FUNCTION_BLOCK FB_PLCTPL_BASE
VAR_INPUT
	{attribute 'OPC.UA.DA':='0'}
	in_sName:				STRING	:= 'Shutter';	// Instance name

	{attribute 'OPC.UA.DA':='0'}
	in_bActiveLowClosed:	BOOL 	:= FALSE;		// If TRUE, the CLOSED signal is Active Low, default FALSE
	{attribute 'OPC.UA.DA':='0'}
	in_bActiveLowFault:		BOOL 	:= FALSE;		// If TRUE, the FAULT signal is Active Low, default FALSE
	{attribute 'OPC.UA.DA':='0'}
	in_bActiveLowOpen:		BOOL 	:= FALSE;		// If TRUE, the OPEN signal is Active Low, default FALSE
	{attribute 'OPC.UA.DA':='0'}
	in_bActiveLowSwitch:	BOOL 	:= FALSE;		// If TRUE, the SWITCH signal is Active Low, default FALSE

	{attribute 'OPC.UA.DA':='0'}
	in_bIgnoreClosed:		BOOL 	:= FALSE;		// If TRUE, the CLOSED signal is Ignored, default FALSE
	{attribute 'OPC.UA.DA':='0'}
	in_bIgnoreFault:		BOOL 	:= FALSE;		// If TRUE, the FAULT signal is Ignored, default FALSE
	{attribute 'OPC.UA.DA':='0'}
	in_bIgnoreOpen:			BOOL 	:= FALSE;		// If TRUE, the OPEN signal is Ignored, default FALSE

	
	{attribute 'OPC.UA.DA':='0'}
	in_bInitialState:		BOOL 	:= FALSE;		// Default shutter position is FALSE/CLOSED
	{attribute 'OPC.UA.DA':='0'}
	in_nTimeout:     		UDINT 	:= 3000;		// Timeout for OPEN/CLOSE transitions [msec], default 3000 ms

	{attribute 'OPC.UA.DA':='0'}
	in_bLogExtTime:			BOOL 	:= FALSE;		// If TRUE, use external time in event logs. Default FALSE.
	{attribute 'OPC.UA.DA':='0'}
	in_bLog:				BOOL 	:= TRUE;		// If TRUE, log events. Default TRUE.
END_VAR
VAR_OUTPUT
END_VAR
VAR RETAIN
END_VAR
VAR
	{attribute 'OPC.UA.DA' := '1'}
	cfg:		T_PLCTPL_CFG;	
	{attribute 'OPC.UA.DA' := '1'}
	ctrl:		T_PLCTPL_CTRL;	
	{attribute 'OPC.UA.DA' := '1'}
	{attribute 'OPC.UA.DA.Access' := '1'}
	info:		T_PLCTPL_INFO;	(* ReadOnly *)
	{attribute 'OPC.UA.DA' := '1'}
	{attribute 'OPC.UA.DA.Access' := '1'}
	stat:		T_PLCTPL_STAT;	(* ReadOnly *)

	{attribute 'OPC.UA.DA' := '0'}
	nEvent:		      	DINT := E_PLCTPL_EVENT.NONE;
	{attribute 'OPC.UA.DA' := '0'}
	nInternalEvent:		DINT := E_PLCTPL_EVENT.NONE;
	
	// Operational Events
	{attribute 'OPC.UA.DA' := '0'}
	fbEventStart:	FB_TcMessage;
	{attribute 'OPC.UA.DA' := '0'}
	fbEventEnd:		FB_TcMessage;
	{attribute 'OPC.UA.DA' := '0'}
	fbEventError:	FB_TcMessage;
	{attribute 'OPC.UA.DA' := '0'}
	fbEventDebug:	FB_TcMessage;
	{attribute 'OPC.UA.DA' := '0'}
	fbEventGeneral:	FB_TcMessage;
	
	(***** Physical signals - to be mapped!!! *****)

	(* Outputs *)

	(* Inputs *)
	
	// Flag if the device is ready to receive commands.
	// It takes a couple of cycles for the system to read inputs after reboot.
	{attribute 'OPC.UA.DA' := '0'}
	bDeviceReady:	BOOL 	:= FALSE;

END_VAR

// On first cycle configure from input params and internally execute M_UserConfigure()
IF NOT bDeviceReady THEN
	// Set device Configuration
	M_Configure();
	RETURN;
END_IF

// Increment counter.
// This will be seen as 'alive' flag.
stat.nCycleCounter	:= stat.nCycleCounter + 1;


(* === Check for commands and internal events to be processed === *)
CheckForEvents();

(* === Process events according to the State Machine === *)
ProcessEvents();

METHOD ActionCloseExecute
VAR_INPUT
END_VAR
END_METHOD

METHOD ActionDisableExecute
VAR_INPUT
END_VAR
END_METHOD

METHOD ActionEnableComplete
VAR_INPUT
END_VAR
END_METHOD

METHOD ActionEnableExecute
VAR_INPUT
END_VAR
END_METHOD

METHOD ActionErrExecute
VAR_INPUT
	nEventId:			DINT;
END_VAR
END_METHOD

METHOD ActionInitAbort
VAR_INPUT
END_VAR
END_METHOD

METHOD ActionInitComplete
VAR_INPUT
END_VAR
END_METHOD

METHOD ActionInitExecute
VAR_INPUT
END_VAR
END_METHOD

METHOD ActionInitReject
VAR_INPUT
END_VAR
END_METHOD

METHOD ActionOpenExecute
VAR_INPUT
END_VAR
END_METHOD

METHOD ActionResetExecute
VAR_INPUT
END_VAR
END_METHOD

METHOD ActionStopExecute
VAR_INPUT
END_VAR
END_METHOD

METHOD ActionUnexpExecute
VAR_INPUT
	nEventId:			DINT;
END_VAR
END_METHOD

METHOD ActivityClosing
VAR_INPUT
END_VAR
END_METHOD

METHOD ActivityDisabling
VAR_INPUT
END_VAR
END_METHOD

METHOD ActivityInitializing
VAR_INPUT
END_VAR
END_METHOD

METHOD ActivityOpening
VAR_INPUT
END_VAR
END_METHOD

METHOD CheckForEvents
VAR_INPUT
END_VAR
END_METHOD

METHOD M_Configure : BOOL
VAR_INPUT
END_VAR
VAR
     fbGetCurTaskIdx:	GETCURTASKINDEX;
END_VAR
// If device is ready, there is nothing to configure.
IF bDeviceReady THEN
	RETURN;
END_IF

// If first cycle, copy configuration AND RETURN in order for the system to read all inputs before doing any work
IF stat.nCycleCounter = 0 THEN
	cfg.sName				:= in_sName;			// Instance name
	cfg.bActiveLowClosed	:= in_bActiveLowClosed;	// If TRUE, the CLOSED signal is Active Low, default FALSE
	cfg.bActiveLowFault		:= in_bActiveLowFault;	// If TRUE, the FAULT signal is Active Low, default FALSE
	cfg.bActiveLowOpen		:= in_bActiveLowOpen;	// If TRUE, the OPEN signal is Active Low, default FALSE
	cfg.bActiveLowSwitch	:= in_bActiveLowSwitch;	// If TRUE, the SWITCH signal is Active Low, default FALSE

	cfg.bIgnoreClosed		:= in_bIgnoreClosed;	// If TRUE, the CLOSED signal is Ignored, default FALSE
	cfg.bIgnoreFault		:= in_bIgnoreFault;		// If TRUE, the FAULT signal is Ignored, default FALSE
	cfg.bIgnoreOpen			:= in_bIgnoreOpen;		// If TRUE, the OPEN signal is Ignored, default FALSE

	cfg.bInitialState		:= in_bInitialState;	// Default shutter position is FALSE/CLOSED
	cfg.nTimeout			:= in_nTimeout;			// Timeout for OPEN/CLOSE transitions [msec], default 3000 ms

	cfg.bLogExtTime			:= in_bLogExtTime;		// If TRUE, use external time in event logs
	cfg.bLog				:= in_bLog;				// If TRUE, use external time in event logs
	
	// Get the version number 
	stat.sLibVersion	:= Global_Version.stLibVersion_ESO_LDC_PLC_Template_Library.sVersion;

 	// Get cycle time in microsec.
	// CycleTime in _TaskInfo is given in 100 ns. 1 us = 1000 ns
	fbGetCurTaskIdx();
	stat.nCycleTime	:=  (TwinCAT_SystemInfoVarList._TaskInfo[fbGetCurTaskIdx.index].CycleTime)/10;
	
	// Increment counter.
	stat.nCycleCounter	:= stat.nCycleCounter + 1;
	RETURN;
ELSIF (stat.nCycleCounter * stat.nCycleTime) < 5000000 THEN
	// EtherCAT is normally ready after 3.5 sec.
	// We give it 5 sec to consider it to be ready.
	// Increment counter.
	stat.nCycleCounter	:= stat.nCycleCounter + 1;
	RETURN;
END_IF

// The system shoud be ready, i.e. coupler state is 8.

// Create Event instances
fbEventStart.CreateEx	(TC_EVENTS.plctplOpsEventClass.ActionStart,0);
fbEventEnd.CreateEx		(TC_EVENTS.plctplOpsEventClass.ActionEnd,0);
fbEventError.CreateEx	(TC_EVENTS.plctplOpsEventClass.Error,0);
fbEventDebug.CreateEx	(TC_EVENTS.plctplOpsEventClass.Debug,0);
fbEventGeneral.CreateEx	(TC_EVENTS.plctplOpsEventClass.General,0);

// The device is ready now.
bDeviceReady := TRUE;


// Clear errors
M_SetStatus(E_PLCTPL_ERROR.OK);
END_METHOD

METHOD M_GetErrorText : STRING
VAR_INPUT
	ErrorCode:	DINT;
END_VAR
VAR
	str:	STRING;
END_VAR
CASE ErrorCode OF
	E_PLCTPL_ERROR.OK:					str	:= 'OK';
	E_PLCTPL_ERROR.HW_NOT_OP:			str	:= 'ERROR: TwinCAT not in OP state or CouplerState not mapped.';
	E_PLCTPL_ERROR.INIT_FAILURE:			str	:= 'ERROR: INIT command aborted due to STOP or RESET.';
	E_PLCTPL_ERROR.UNEXPECTED_CLOSED:	str	:= 'ERROR: Shutter unexpectedly closed.';
	E_PLCTPL_ERROR.UNEXPECTED_NONE:		str	:= 'ERROR: Unexpectedly no OPEN or CLOSED signal active.';
	E_PLCTPL_ERROR.UNEXPECTED_OPENED:	str	:= 'ERROR: Shutter unexpectedly opened.';
	E_PLCTPL_ERROR.FAULT_SIG:			str	:= 'ERROR: Fault signal active.';
	E_PLCTPL_ERROR.BOTH_SIG_ACTIVE:		str	:= 'ERROR: Both OPEN and CLOSED signals active.';
	E_PLCTPL_ERROR.TIMEOUT_ENABLE:		str	:= 'ERROR: ENABLE timed out.';
	E_PLCTPL_ERROR.TIMEOUT_DISABLE:		str	:= 'ERROR: DISABLE timed out.';
	E_PLCTPL_ERROR.TIMEOUT_INIT:			str	:= 'ERROR: INIT timed out.';
	E_PLCTPL_ERROR.TIMEOUT_CLOSE:		str	:= 'ERROR: CLOSE timed out.';
	E_PLCTPL_ERROR.TIMEOUT_OPEN:			str	:= 'ERROR: OPEN timed out.';
	E_PLCTPL_ERROR.SIM_NOT_INITIALISED:	str	:= 'ERROR: Shutter simulator not initialised.';
	E_PLCTPL_ERROR.SIM_NULL_POINTER:		str	:= 'ERROR: NULL pointer to Shutter.';
ELSE
	str	:= 'Unregistered error.';
END_CASE

M_GetErrorText	:= str;
END_METHOD

METHOD M_LogEventDebug : BOOL
VAR_INPUT
	sText:	STRING	:= '';
END_VAR
// Log Debug events only if both logging and debugging is enabled
IF cfg.bLog AND cfg.bDebug THEN
	fbEventDebug.ipArguments.Clear().AddString(sText);
	fbEventDebug.Send(0);
END_IF
END_METHOD

METHOD M_LogEventEnd : BOOL
VAR_INPUT
	sText:	STRING	:= '';
END_VAR
// Log only if logging is enabled
IF  NOT cfg.bLog THEN
	RETURN;
END_IF

fbEventEnd.ipArguments.Clear().AddString(sText);
fbEventEnd.Send(0);
END_METHOD

METHOD M_LogEventError : BOOL
VAR_INPUT
	sText:	STRING	:= '';
END_VAR
// Log only if logging is enabled
IF  NOT cfg.bLog THEN
	RETURN;
END_IF

fbEventError.ipArguments.Clear().AddString(sText);
fbEventError.Send(0);
END_METHOD

METHOD M_LogEventGeneral : BOOL
VAR_INPUT
	sText:	STRING	:= '';
END_VAR
// Log only if logging is enabled
IF  NOT cfg.bLog THEN
	RETURN;
END_IF

fbEventGeneral.ipArguments.Clear().AddString(sText);
fbEventGeneral.Send(0);
END_METHOD

METHOD M_LogEventStart : BOOL
VAR_INPUT
	sText:	STRING	:= '';
END_VAR
// Log only if logging is enabled
IF  NOT cfg.bLog THEN
	RETURN;
END_IF

fbEventStart.ipArguments.Clear().AddString(sText);
fbEventStart.Send(0);
END_METHOD

METHOD M_SetStatus
VAR_INPUT
	nErrorCode:	E_PLCTPL_ERROR;
END_VAR
stat.nErrorCode 	:= nErrorCode;
stat.sErrorText 	:= M_GetErrorText(nErrorCode);

IF nErrorCode <> E_PLCTPL_ERROR.OK THEN
	stat.sStatus	:= 'ERROR';
	stat.nStatus	:= E_PLCTPL_STATUS.ERROR;
ELSE
	stat.sStatus	:= 'OK';
	stat.nStatus	:= E_PLCTPL_STATUS.OK;
END_IF
END_METHOD

METHOD ProcessEvents
VAR_INPUT
END_VAR

VAR
	ActionUnexpectedOpenExecute: INT;
END_VAR

(* 
	Before processing the event, execute the Do-Activity tasks. 
	Note that, in case of orthogonal regions, more than one Do-Activity 
	could run in the same PLC cycle.
	Note: Most of these activities have timeouts since they take time.
*)

IF stat.nSubstate = E_PLCTPL_SUBSTATE.NOTOP_INITIALIZING THEN
	ActivityInitializing();
END_IF

IF stat.nSubstate = E_PLCTPL_SUBSTATE.OP_OPENING THEN
	ActivityOpening();
END_IF

IF stat.nSubstate = E_PLCTPL_SUBSTATE.OP_CLOSING THEN
	ActivityClosing();
END_IF

IF stat.nSubstate = E_PLCTPL_SUBSTATE.OP_DISABLING THEN
	ActivityDisabling();
END_IF


(* 
	Evaluate state machine transitions.
*)

CASE stat.nState OF

//***********************************
// NOTOP
//***********************************
E_PLCTPL_STATE.NOTOP:

	(* Transitions from NOTOP substates *)
	CASE stat.nSubstate OF
	
	E_PLCTPL_SUBSTATE.NOTOP_NOTREADY:		
		IF nEvent = E_PLCTPL_EVENT.INIT THEN
			ActionInitExecute();
			SetState(E_PLCTPL_STATE.NOTOP, E_PLCTPL_SUBSTATE.NOTOP_INITIALIZING);
			M_SetStatus(E_PLCTPL_ERROR.OK);
			RETURN;
		END_IF
		
	E_PLCTPL_SUBSTATE.NOTOP_INITIALIZING:			
		IF nEvent = E_PLCTPL_EVENT.STOP THEN
			ActionInitAbort();
			SetState(E_PLCTPL_STATE.NOTOP, E_PLCTPL_SUBSTATE.NOTOP_NOTREADY);
			RETURN;
		ELSIF nEvent = E_PLCTPL_EVENT.ERRINIT THEN
			SetState(E_PLCTPL_STATE.NOTOP, E_PLCTPL_SUBSTATE.NOTOP_ERROR);
			RETURN;
		ELSIF nEvent = E_PLCTPL_EVENT.INITCLOSED THEN
			ActionInitComplete();
			SetState(E_PLCTPL_STATE.NOTOP, E_PLCTPL_SUBSTATE.NOTOP_READY_CLOSED);
			RETURN;
		ELSIF nEvent = E_PLCTPL_EVENT.INITOPEN THEN
			ActionInitComplete();
			SetState(E_PLCTPL_STATE.NOTOP, E_PLCTPL_SUBSTATE.NOTOP_READY_OPEN);
			RETURN;
		END_IF
		
	E_PLCTPL_SUBSTATE.NOTOP_READY_CLOSED:			
		IF nEvent = E_PLCTPL_EVENT.ISOPEN THEN
			ActionUnexpExecute(nEvent);
			SetState(E_PLCTPL_STATE.NOTOP, E_PLCTPL_SUBSTATE.NOTOP_READY_OPEN);
			RETURN;
		ELSIF nEvent = E_PLCTPL_EVENT.ENABLE THEN
			ActionEnableComplete();
			SetState(E_PLCTPL_STATE.OP, E_PLCTPL_SUBSTATE.OP_CLOSED);
			RETURN;
		END_IF

	E_PLCTPL_SUBSTATE.NOTOP_READY_OPEN:			
		IF nEvent = E_PLCTPL_EVENT.ISCLOSED THEN
			ActionUnexpExecute(nEvent);
			SetState(E_PLCTPL_STATE.NOTOP, E_PLCTPL_SUBSTATE.NOTOP_READY_CLOSED);
			RETURN;
		ELSIF nEvent = E_PLCTPL_EVENT.ENABLE THEN
			ActionEnableComplete();
			SetState(E_PLCTPL_STATE.OP, E_PLCTPL_SUBSTATE.OP_OPEN);
			RETURN;
		END_IF

	E_PLCTPL_SUBSTATE.NOTOP_ERROR:			
		IF	nEvent = E_PLCTPL_EVENT.HWOK 				AND 
			stat.nErrorCode = E_PLCTPL_ERROR.HW_NOT_OP 	THEN
			SetState(E_PLCTPL_STATE.NOTOP, E_PLCTPL_SUBSTATE.NOTOP_NOTREADY);
			RETURN;
		END_IF
		
	END_CASE

	(* Transitions from NOTOP state *)
	IF nEvent = E_PLCTPL_EVENT.ERRHW THEN
		SetState(E_PLCTPL_STATE.NOTOP, E_PLCTPL_SUBSTATE.NOTOP_ERROR);
		RETURN;
	ELSIF nEvent = E_PLCTPL_EVENT.ERRFAULT THEN
		// TODO
		SetState(E_PLCTPL_STATE.NOTOP, E_PLCTPL_SUBSTATE.NOTOP_ERROR);			
		RETURN;
	ELSIF nEvent = E_PLCTPL_EVENT.ERRALLACTIVE THEN
		// TODO
		ActionErrExecute(nEvent);
		SetState(E_PLCTPL_STATE.NOTOP, E_PLCTPL_SUBSTATE.NOTOP_ERROR);
		RETURN;
	END_IF
	
//***********************************
// OPERATIONAL
//***********************************
E_PLCTPL_STATE.OP:

	(* Transitions from OP subastates *)
	CASE stat.nSubstate OF
	E_PLCTPL_SUBSTATE.OP_CLOSED:			
		IF nEvent = E_PLCTPL_EVENT.OPEN THEN
			ActionOpenExecute();
			SetState(E_PLCTPL_STATE.OP, E_PLCTPL_SUBSTATE.OP_OPENING);
			RETURN;
		ELSIF nEvent = E_PLCTPL_EVENT.CLOSE THEN
			// Nothing to do. Just clear previous error, if any.
			M_SetStatus(E_PLCTPL_ERROR.OK);
			RETURN;
		ELSIF nEvent = E_PLCTPL_EVENT.ISOPEN THEN
			ActionUnexpExecute(nEvent);
			SetState(E_PLCTPL_STATE.OP, E_PLCTPL_SUBSTATE.OP_OPEN);
			RETURN;
		ELSIF nEvent = E_PLCTPL_EVENT.DISABLE THEN
			ActionDisableExecute();
			SetState(E_PLCTPL_STATE.OP, E_PLCTPL_SUBSTATE.OP_DISABLING);
			RETURN;		
		ELSIF nEvent = E_PLCTPL_EVENT.ERRNONEACTIVE THEN
			ActionUnexpExecute(nEvent);
			SetState(E_PLCTPL_STATE.OP, E_PLCTPL_SUBSTATE.OP_ERROR);
			RETURN;				
		END_IF

	E_PLCTPL_SUBSTATE.OP_OPENING:			
		IF nEvent = E_PLCTPL_EVENT.ISOPEN THEN
			SetState(E_PLCTPL_STATE.OP, E_PLCTPL_SUBSTATE.OP_OPEN);
			RETURN;
		ELSIF nEvent = E_PLCTPL_EVENT.ISCLOSED THEN
			ActionUnexpExecute(nEvent);
			SetState(E_PLCTPL_STATE.OP, E_PLCTPL_SUBSTATE.OP_ERROR);
			RETURN;
		ELSIF nEvent = E_PLCTPL_EVENT.ERRTIMEOUTOPEN THEN
			SetState(E_PLCTPL_STATE.OP, E_PLCTPL_SUBSTATE.OP_ERROR);
			RETURN;
		ELSIF nEvent = E_PLCTPL_EVENT.STOP THEN
			ActionStopExecute();
			SetState(E_PLCTPL_STATE.OP, E_PLCTPL_SUBSTATE.OP_CLOSING);
			RETURN;			
		END_IF
		
	E_PLCTPL_SUBSTATE.OP_OPEN:			
		IF nEvent = E_PLCTPL_EVENT.CLOSE THEN
			ActionCloseExecute();
			SetState(E_PLCTPL_STATE.OP, E_PLCTPL_SUBSTATE.OP_CLOSING);
			RETURN;
		ELSIF nEvent = E_PLCTPL_EVENT.OPEN THEN
			// Nothing to do. Just clear previous error, if any.
			M_SetStatus(E_PLCTPL_ERROR.OK);
			RETURN;
		ELSIF nEvent = E_PLCTPL_EVENT.ISCLOSED THEN
			ActionUnexpExecute(nEvent);
			SetState(E_PLCTPL_STATE.OP, E_PLCTPL_SUBSTATE.OP_CLOSED);
			RETURN;
		ELSIF nEvent = E_PLCTPL_EVENT.DISABLE THEN
			ActionDisableExecute();
			SetState(E_PLCTPL_STATE.OP, E_PLCTPL_SUBSTATE.OP_DISABLING);
			RETURN;	
		ELSIF nEvent = E_PLCTPL_EVENT.ERRNONEACTIVE THEN
			ActionUnexpExecute(nEvent);
			SetState(E_PLCTPL_STATE.OP, E_PLCTPL_SUBSTATE.OP_ERROR);
			RETURN;				
		END_IF
		
	E_PLCTPL_SUBSTATE.OP_CLOSING:			
		IF nEvent = E_PLCTPL_EVENT.ISCLOSED THEN
			SetState(E_PLCTPL_STATE.OP, E_PLCTPL_SUBSTATE.OP_CLOSED);
			RETURN;
		ELSIF nEvent = E_PLCTPL_EVENT.ISOPEN THEN
			SetState(E_PLCTPL_STATE.OP, E_PLCTPL_SUBSTATE.OP_OPEN);
			RETURN;
		ELSIF nEvent = E_PLCTPL_EVENT.ERRTIMEOUTCLOSE THEN
			SetState(E_PLCTPL_STATE.OP, E_PLCTPL_SUBSTATE.OP_ERROR);
			RETURN;
		ELSIF nEvent = E_PLCTPL_EVENT.STOP THEN
			ActionStopExecute();
			SetState(E_PLCTPL_STATE.OP, E_PLCTPL_SUBSTATE.OP_OPENING);
			RETURN;			
		END_IF
		
	E_PLCTPL_SUBSTATE.OP_ERROR:			
		IF nEvent = E_PLCTPL_EVENT.CLOSE THEN
			ActionCloseExecute();
			SetState(E_PLCTPL_STATE.OP, E_PLCTPL_SUBSTATE.OP_CLOSING);
			RETURN;
		ELSIF nEvent = E_PLCTPL_EVENT.OPEN THEN
			ActionOpenExecute();
			SetState(E_PLCTPL_STATE.OP, E_PLCTPL_SUBSTATE.OP_OPENING);
			RETURN;			
		ELSIF nEvent = E_PLCTPL_EVENT.ISOPEN THEN
			M_LogEventGeneral('Recovered from error. Shutter is OPEN.');
			SetState(E_PLCTPL_STATE.OP, E_PLCTPL_SUBSTATE.OP_OPEN);
			RETURN;			
		ELSIF nEvent = E_PLCTPL_EVENT.ISCLOSED THEN
			M_LogEventGeneral('Recovered from error. Shutter is CLOSED.');
			SetState(E_PLCTPL_STATE.OP, E_PLCTPL_SUBSTATE.OP_CLOSED);
			RETURN;	
		ELSIF nEvent = E_PLCTPL_EVENT.DISABLE THEN
			SetState(E_PLCTPL_STATE.OP, E_PLCTPL_SUBSTATE.OP_DISABLING);
			RETURN;			
		END_IF

	E_PLCTPL_SUBSTATE.OP_DISABLING:			
		IF nEvent = E_PLCTPL_EVENT.DISABLECLOSED THEN
			SetState(E_PLCTPL_STATE.NOTOP, E_PLCTPL_SUBSTATE.NOTOP_READY_CLOSED);
			RETURN;
		ELSIF nEvent = E_PLCTPL_EVENT.DISABLEOPEN THEN
			SetState(E_PLCTPL_STATE.NOTOP, E_PLCTPL_SUBSTATE.NOTOP_READY_OPEN);
			RETURN;
		ELSIF nEvent = E_PLCTPL_EVENT.ERRDISABLE THEN
			SetState(E_PLCTPL_STATE.OP, E_PLCTPL_SUBSTATE.OP_ERROR);
			RETURN;
		END_IF
		
	END_CASE
	
	(* Transitions from OP state *)
	IF nEvent = E_PLCTPL_EVENT.ERRHW THEN
		SetState(E_PLCTPL_STATE.OP, E_PLCTPL_SUBSTATE.OP_ERROR);
		RETURN;
	ELSIF nEvent = E_PLCTPL_EVENT.ERRFAULT THEN
		SetState(E_PLCTPL_STATE.OP, E_PLCTPL_SUBSTATE.OP_ERROR);
		RETURN;
	ELSIF nEvent = E_PLCTPL_EVENT.ERRALLACTIVE THEN
		// TODO
		ActionErrExecute(nEvent);
		SetState(E_PLCTPL_STATE.OP, E_PLCTPL_SUBSTATE.OP_ERROR);
		RETURN;
	END_IF
	
END_CASE

(* 
	"Global" internal transitions valid in any state should go here.
	They do not change the active state configuration. 
	They are evaluated after all the others transitions have been 
	considered.
*) 
IF nEvent = E_PLCTPL_EVENT.RESET THEN
	ActionResetExecute();
	SetState(E_PLCTPL_STATE.NOTOP, E_PLCTPL_SUBSTATE.NOTOP_NOTREADY);
	RETURN;
END_IF
END_METHOD

METHOD SetAction
VAR_INPUT
	actionName:		STRING;
END_VAR


stat.sActionDesc := actionName;
END_METHOD

METHOD SetEvent
VAR_INPUT
	nEventId:			DINT;
END_VAR

nEvent := nEventId;

CASE nEventId OF
	E_PLCTPL_EVENT.NONE:
		stat.sEventDesc := '';
		RETURN;
		
	E_PLCTPL_EVENT.RESET:
		stat.sEventDesc := 'CMD RESET';
		RETURN;
	
	E_PLCTPL_EVENT.INIT:
		stat.sEventDesc := 'CMD INIT';
		RETURN;

	E_PLCTPL_EVENT.STOP:
		stat.sEventDesc := 'CMD STOP';
		RETURN;

	E_PLCTPL_EVENT.ENABLE:
		stat.sEventDesc := 'CMD ENABLE';
		RETURN;

	E_PLCTPL_EVENT.DISABLE:
		stat.sEventDesc := 'CMD DISABLE';
		RETURN;

	E_PLCTPL_EVENT.OPEN:
		stat.sEventDesc := 'CMD OPEN';
		RETURN;

	E_PLCTPL_EVENT.CLOSE:
		stat.sEventDesc := 'CMD CLOSE';
		RETURN;
	
	(* events corresponding to internal events *)
	E_PLCTPL_EVENT.INITCLOSED:
		stat.sEventDesc := 'INT INITCLOSED';
		RETURN;

	E_PLCTPL_EVENT.INITOPEN:
		stat.sEventDesc := 'INT INITOPEN';
		RETURN;

	E_PLCTPL_EVENT.DISABLECLOSED:
		stat.sEventDesc := 'INT DISABLECLOSED';
		RETURN;
	
	E_PLCTPL_EVENT.DISABLEOPEN:
		stat.sEventDesc := 'INT DISABLEOPEN';
		RETURN;
	
	(* evetnts mapped to HW signals *)
	E_PLCTPL_EVENT.ISOPEN:
		stat.sEventDesc := 'SIG ISOPEN';
		RETURN;

	E_PLCTPL_EVENT.ISCLOSED:
		stat.sEventDesc := 'SIG ISCLOSED';
		RETURN;

	E_PLCTPL_EVENT.HWOK:
		stat.sEventDesc := 'SIG HWOK';
		RETURN;

	E_PLCTPL_EVENT.ERRHW:
		stat.sEventDesc := 'INT ERRHW';
		RETURN;

	E_PLCTPL_EVENT.ERRFAULT:	
		stat.sEventDesc := 'INT ERRFAULT';
		RETURN;

	E_PLCTPL_EVENT.ERRALLACTIVE:
		stat.sEventDesc := 'INT ERRALLACTIVE';
		RETURN;
	
	E_PLCTPL_EVENT.ERRNONEACTIVE:	
		stat.sEventDesc := 'INT ERRNONEACTIVE';
		RETURN;
		
	E_PLCTPL_EVENT.ERRINIT:
		stat.sEventDesc := 'INT ERRINIT';
		RETURN;

	E_PLCTPL_EVENT.ERRDISABLE:
		stat.sEventDesc := 'INT ERRDISABLE';
		RETURN;
	
END_CASE 

(* INTERNAL ERROR *)
stat.sEventDesc := 'UNKNOWN EVENT';
END_METHOD

METHOD SetState : BOOL
VAR_INPUT
	nState:			E_PLCTPL_STATE;
	nSubstate:		E_PLCTPL_SUBSTATE;
END_VAR
(* 
	Update State Machine active state configuration.

	ToDo: support initial pseudo state/substate.
*)

IF nState <> E_PLCTPL_STATE.NONE THEN
	stat.nState	:= nState;
END_IF
IF nSubstate <> E_PLCTPL_SUBSTATE.NONE THEN
	stat.nSubstate	:= nSubstate;
END_IF

(* Update active state configuration description *)

IF nState = E_PLCTPL_STATE.NOTOP THEN
	stat.sState	:= 'NOT OP';
ELSIF nState = E_PLCTPL_STATE.OP THEN
	stat.sState	:= 'OPERATIONAL';
END_IF

IF nSubstate = E_PLCTPL_SUBSTATE.NOTOP_NOTREADY THEN
	stat.sSubstate	:= 'NOT READY';
ELSIF nSubstate = E_PLCTPL_SUBSTATE.NOTOP_INITIALIZING THEN
	stat.sSubstate	:= 'INITIALIAZING';
ELSIF nSubstate = E_PLCTPL_SUBSTATE.NOTOP_READY_CLOSED THEN
	stat.sSubstate	:= 'READY CLOSED';
ELSIF nSubstate = E_PLCTPL_SUBSTATE.NOTOP_READY_OPEN THEN
	stat.sSubstate	:= 'READY OPEN';
ELSIF nSubstate = E_PLCTPL_SUBSTATE.NOTOP_ERROR THEN
	stat.sSubstate	:= 'ERROR';
ELSIF nSubstate = E_PLCTPL_SUBSTATE.OP_CLOSED THEN
	stat.sSubstate	:= 'CLOSED';
ELSIF nSubstate = E_PLCTPL_SUBSTATE.OP_OPEN THEN
	stat.sSubstate	:= 'OPEN';
ELSIF nSubstate = E_PLCTPL_SUBSTATE.OP_CLOSING THEN
	stat.sSubstate	:= 'CLOSING';
ELSIF nSubstate = E_PLCTPL_SUBSTATE.OP_OPENING THEN
	stat.sSubstate	:= 'OPENING';
ELSIF nSubstate = E_PLCTPL_SUBSTATE.OP_DISABLING THEN
	stat.sSubstate	:= 'DISABLING';
ELSIF nSubstate = E_PLCTPL_SUBSTATE.OP_ERROR THEN
	stat.sSubstate	:= 'ERROR';
ELSE
	stat.sSubstate	:= '';
END_IF


SetState	:= TRUE;
END_METHOD

END_FUNCTION_BLOCK

(* stored: Version 1.1.0.1, ProductVersion 3.1.4024.9
   POU FB_PLCTPL_BASE: Id {9b20579e-46f1-487a-b0e9-71610139463f}, SpecialFunc None
   Method ActionCloseExecute: Id {8df5e8e5-d231-47e0-80a7-3f3129f3904a}
   Method ActionDisableExecute: Id {6fc35504-cac0-44ac-ad71-a249e896f4d1}
   Method ActionEnableComplete: Id {d3a5feb5-11d8-407c-9384-7da066c05c39}
   Method ActionEnableExecute: Id {ef01bce1-e3d5-44f4-9ac2-7266aba2948c}
   Method ActionErrExecute: Id {f0b03128-67d1-4f29-8bef-9e922ed95113}
   Method ActionInitAbort: Id {e9720cce-33ed-44ab-8765-59705f455dbf}
   Method ActionInitComplete: Id {56051acc-d213-4084-b91c-4495ca171c5d}
   Method ActionInitExecute: Id {7c08ae8b-b17b-4fe9-92ef-38c23e0bebc2}
   Method ActionInitReject: Id {6e09029d-40c6-4972-a65b-1d11fa327959}
   Method ActionOpenExecute: Id {7e32a4c6-40e9-4483-ae7a-330aeaa799ea}
   Method ActionResetExecute: Id {ed28dfa9-8c19-4ef7-b6fa-7e3c1a84e955}
   Method ActionStopExecute: Id {347b68cf-22e4-4432-9e4d-428120ff0276}
   Method ActionUnexpExecute: Id {fabeea70-ef5f-4c6d-b939-031dc980b796}
   Method ActivityClosing: Id {3cce3bbc-fede-4b68-bbe0-e7ac26348c76}
   Method ActivityDisabling: Id {d4f82c1d-d70f-4b02-b15f-63975ee2a792}
   Method ActivityInitializing: Id {8b8e1bac-980c-4f00-b852-db89d34da7dd}
   Method ActivityOpening: Id {1228c683-5117-4fbc-a2ed-13fdab0adf28}
   Method CheckForEvents: Id {21796d32-c062-4e31-afea-506812fda30e}
   Method M_Configure: Id {bd336feb-f03a-429f-92a9-35a747dfe0f6}
   Method M_GetErrorText: Id {8c7cc3da-ad51-4e6b-91f6-ad6e3a854aff}
   Method M_LogEventDebug: Id {76ff400f-eecc-453d-bdbd-16ea83a14a8b}
   Method M_LogEventEnd: Id {924a63d8-c4db-4990-833d-29094815b171}
   Method M_LogEventError: Id {09811c01-7dc5-4d6f-9199-d2731ce1b7ee}
   Method M_LogEventGeneral: Id {a9dfeb89-9fc4-4c54-af42-3043d81bb670}
   Method M_LogEventStart: Id {3bae18c2-756c-4d13-9096-9ce29d4d65af}
   Method M_SetStatus: Id {3c05461c-82e3-4012-8ec1-1b295a1d1d1a}
   Method ProcessEvents: Id {6e9c6b9a-4c2b-4268-a28e-d15cd6e7df03}
   Method SetAction: Id {2acba3b2-45b6-4a2a-b462-51ba88d57ca8}
   Method SetEvent: Id {6b68da34-70da-405a-b0a8-7235e5482c8e}
   Method SetState: Id {725c2510-95cb-4885-9251-304ab558f2e2} *)
